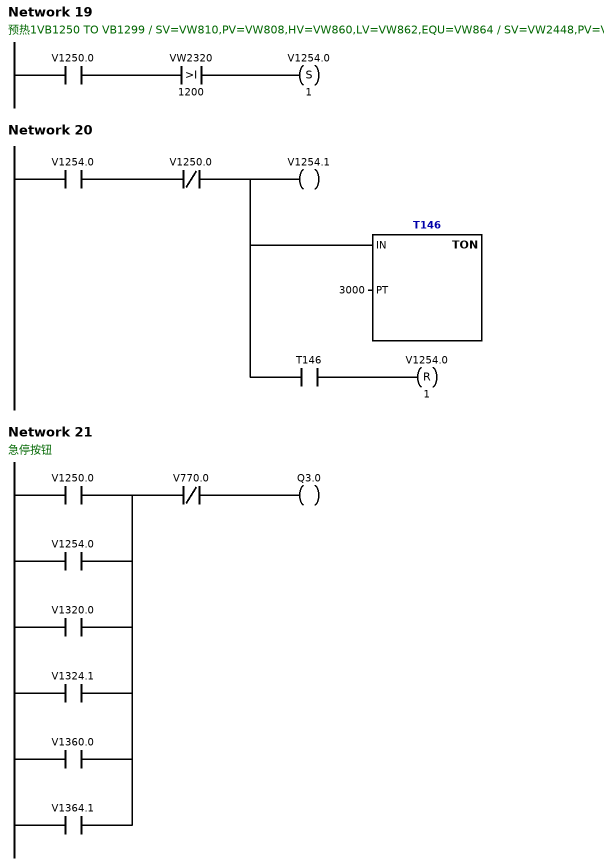
[picture p24: SBR4 networks 19-21]
Network 19
// 预热1VB1250 TO VB1299
// SV=VW810,PV=VW808,HV=VW860,LV=VW862,EQU=VW864
// SV=VW2448,PV=VW2320,HV=VW860,LV=VW862,EQU=VW864
// PV=VW2320 > 120 度就要冷却循环风关机
LD     V1250.0
AW>    VW2320, 1200
S      V1254.0, 1
Network 20
LD     V1254.0
AN     V1250.0
=      V1254.1
TON    T146, 3000
A      T146
R      V1254.0, 1
Network 21
// 急停按钮
LD     V1250.0
O      V1254.0
O      V1320.0
O      V1324.1
O      V1360.0
O      V1364.1
AN     V770.0
=      Q3.0
END_SUBROUTINE_BLOCK

SUBROUTINE_BLOCK WaveSpewWagVB1300_1319:SBR5
TITLE=WaveSpewWagVB1300_1319//T160_T164
BEGIN
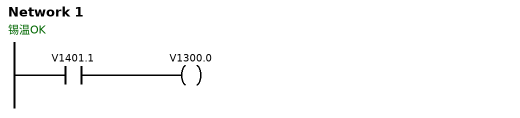
Network 1
// 锡温OK
LD     V1401.1
=      V1300.0
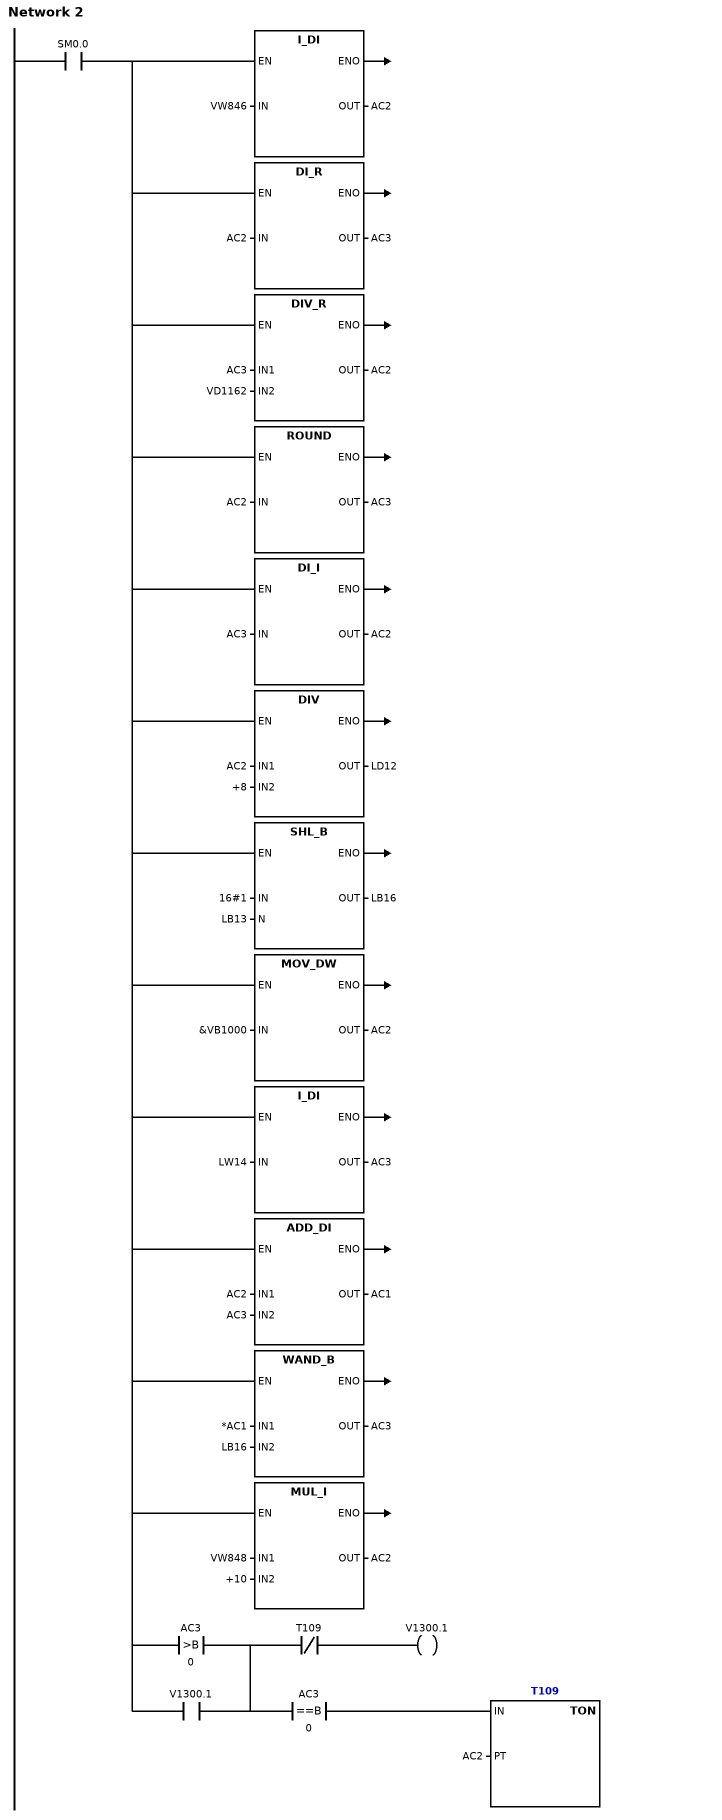
Network 2
LD     SM0.0
ITD    VW846, AC2
DTR    AC2, AC3
MOVR   AC3, AC2
/R     VD1162, AC2
ROUND  AC2, AC3
DTI    AC3, AC2
MOVW   AC2, LW14
DIV    +8, LD12
MOVB   16#1, LB16
SLB    LB16, LB13
MOVD   &VB1000, AC2
ITD    LW14, AC3
MOVD   AC2, AC1
+D     AC3, AC1
MOVB   *AC1, AC3
ANDB   LB16, AC3
MOVW   VW848, AC2
*I     +10, AC2
LDB>   AC3, 0
O      V1300.1
ALD
LPS
AN     T109
=      V1300.1
LPP
AB=    AC3, 0
TON    T109, AC2
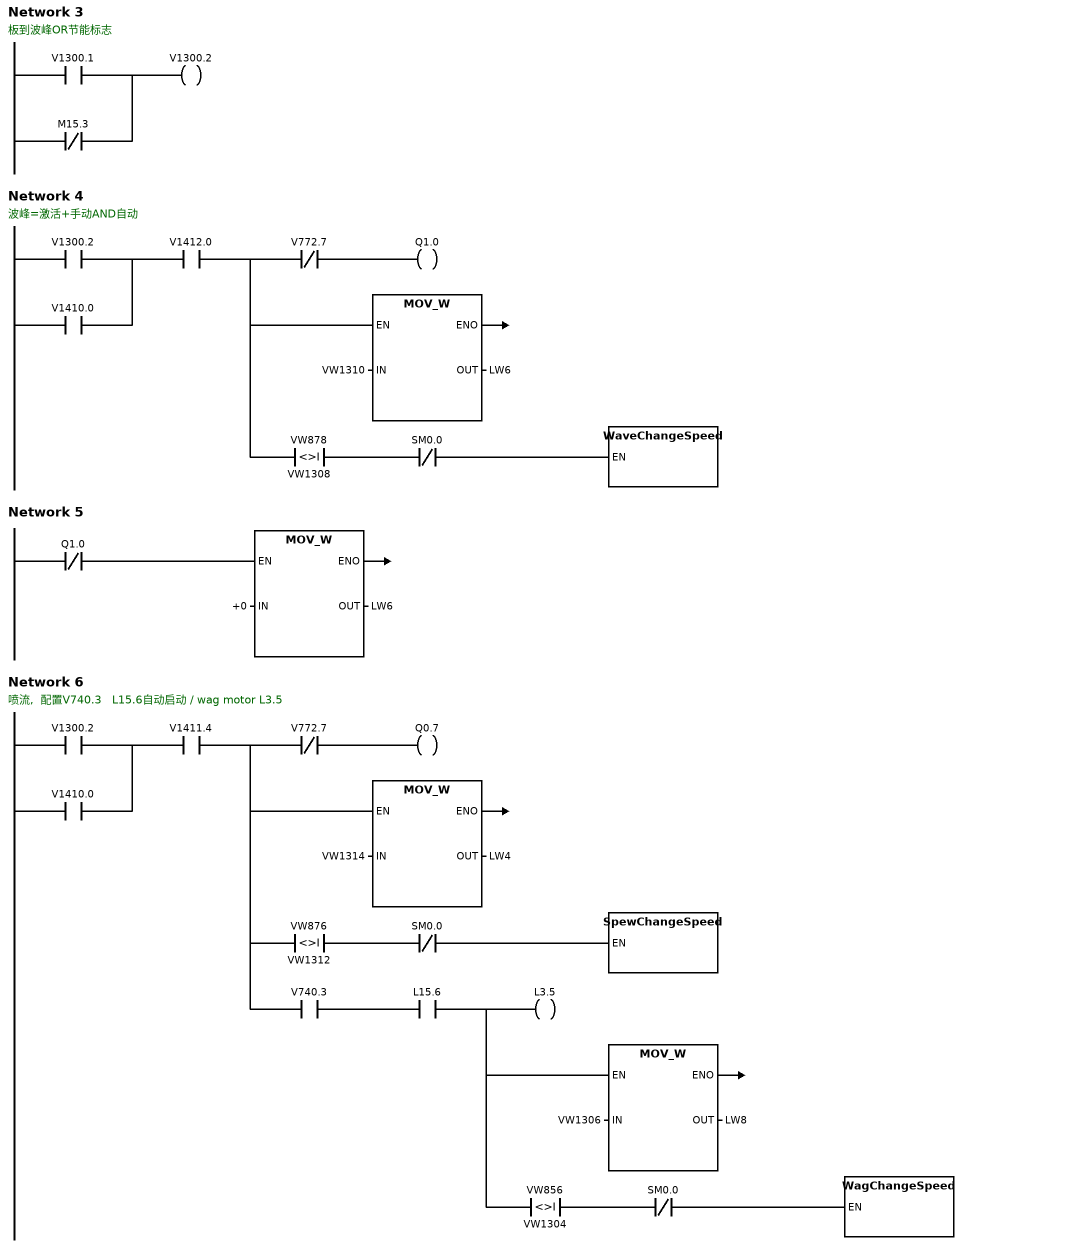
Network 3
// 板到波峰OR节能标志
LD     V1300.1
ON     M15.3
=      V1300.2
Network 4
// 波峰=激活+手动AND自动
LD     V1300.2
O      V1410.0
A      V1412.0
LPS
AN     V772.7
=      Q1.0
LRD
MOVW   VW1310, LW6
LPP
AW<>   VW878, VW1308
AN     SM0.0
CALL   WaveChangeSpeed:SBR23
Network 5
LDN    Q1.0
MOVW   +0, LW6
Network 6
// 喷流,  配置V740.3   L15.6自动启动
// wag motor L3.5
LD     V1300.2
O      V1410.0
A      V1411.4
LPS
AN     V772.7
=      Q0.7
LRD
MOVW   VW1314, LW4
LRD
AW<>   VW876, VW1312
AN     SM0.0
CALL   SpewChangeSpeed:SBR24
LPP
A      V740.3
A      L15.6
=      L3.5
MOVW   VW1306, LW8
AW<>   VW856, VW1304
AN     SM0.0
CALL   WagChangeSpeed:SBR22
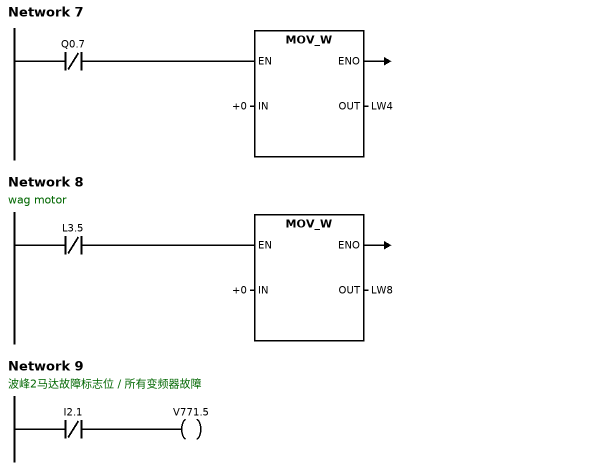
Network 7
LDN    Q0.7
MOVW   +0, LW4
Network 8
// wag motor 
LDN    L3.5
MOVW   +0, LW8
Network 9
// 波峰2马达故障标志位
// 所有变频器故障
LDN    I2.1
=      V771.5
Network 10
// 只要你配置了,喷流就可能产生故障标志位
Network 11
// 只要你配置了,摇动就可能产生故障标志位
END_SUBROUTINE_BLOCK

SUBROUTINE_BLOCK Preheat2VB1320_1359:SBR6
TITLE=
BEGIN
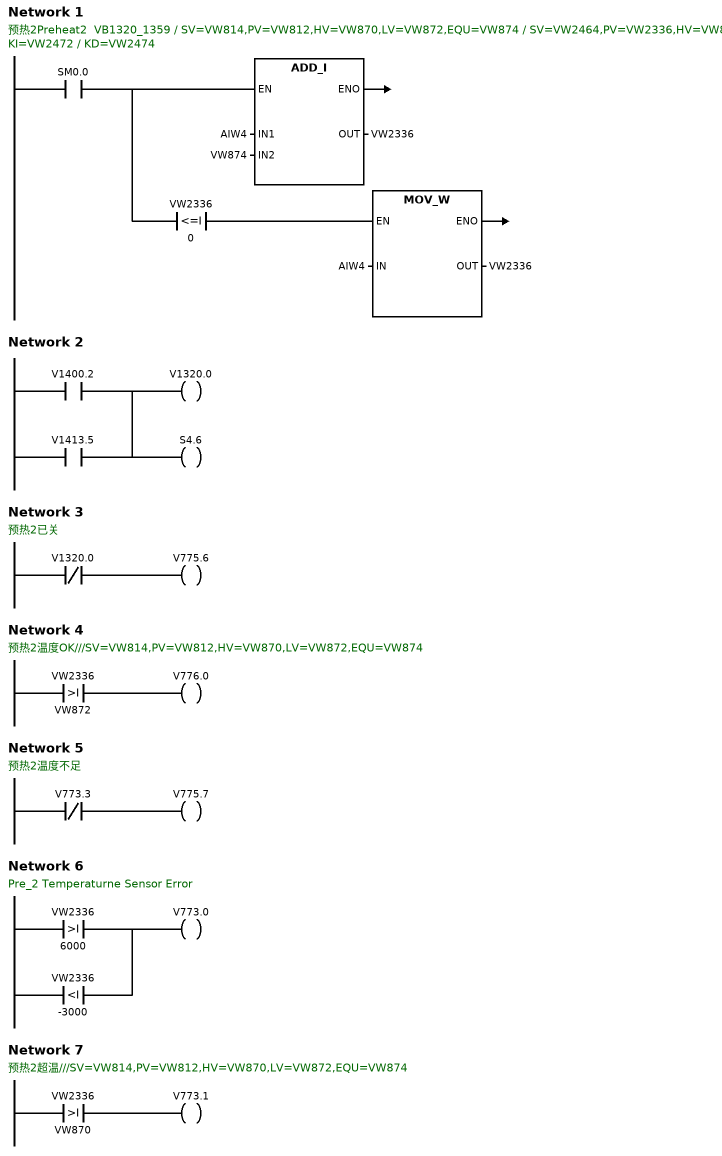
Network 1
// 预热2Preheat2  VB1320_1359
// SV=VW814,PV=VW812,HV=VW870,LV=VW872,EQU=VW874
// SV=VW2464,PV=VW2336,HV=VW870,LV=VW872,EQU=VW874
// 
// KT=VW2468
// KP=VW2470
// KI=VW2472
// KD=VW2474
LD     SM0.0
MOVW   AIW4, VW2336
+I     VW874, VW2336
AW<=   VW2336, 0
MOVW   AIW4, VW2336
Network 2
LD     V1400.2
O      V1413.5
=      V1320.0
=      S4.6
Network 3
// 预热2已关
LDN    V1320.0
=      V775.6
Network 4
// 预热2温度OK///SV=VW814,PV=VW812,HV=VW870,LV=VW872,EQU=VW874
LDW>   VW2336, VW872
=      V776.0
Network 5
// 预热2温度不足
LDN    V773.3
=      V775.7
Network 6
// Pre_2 Temperaturne Sensor Error
LDW>   VW2336, 6000
OW<    VW2336, -3000
=      V773.0
Network 7
// 预热2超温///SV=VW814,PV=VW812,HV=VW870,LV=VW872,EQU=VW874
LDW>   VW2336, VW870
=      V773.1
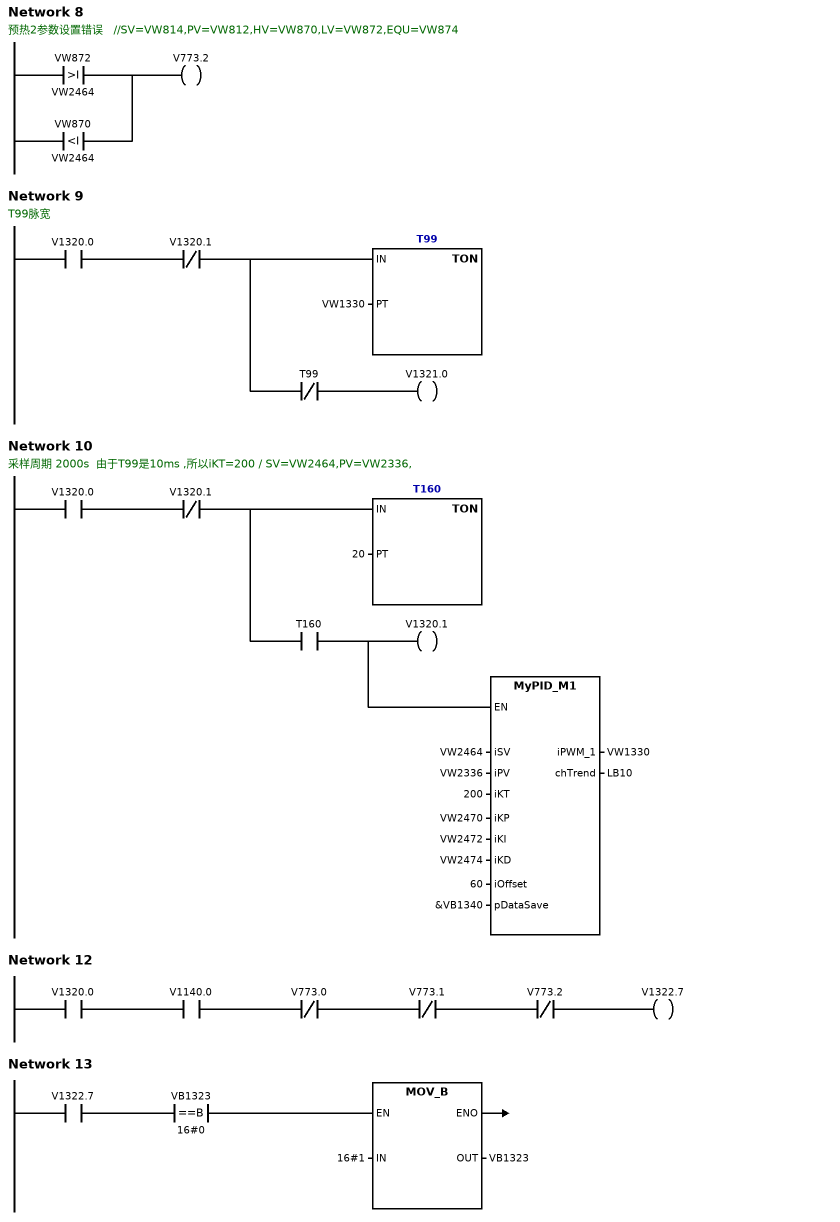
Network 8
// 预热2参数设置错误   //SV=VW814,PV=VW812,HV=VW870,LV=VW872,EQU=VW874
LDW>   VW872, VW2464
OW<    VW870, VW2464
=      V773.2
Network 9
// T99脉宽
LD     V1320.0
AN     V1320.1
TON    T99, VW1330
AN     T99
=      V1321.0
Network 10
// 采样周期 2000s  由于T99是10ms ,所以iKT=200
// SV=VW2464,PV=VW2336,
LD     V1320.0
AN     V1320.1
TON    T160, 20
A      T160
=      V1320.1
CALL   MyPID_M1:SBR30, VW2464, VW2336, 200, VW2470, VW2472, VW2474, 60, &VB1340, VW1330, LB10
Network 12
LD     V1320.0
A      V1140.0
AN     V773.0
AN     V773.1
AN     V773.2
=      V1322.7
Network 13
LD     V1322.7
AB=    VB1323, 16#0
MOVB   16#1, VB1323
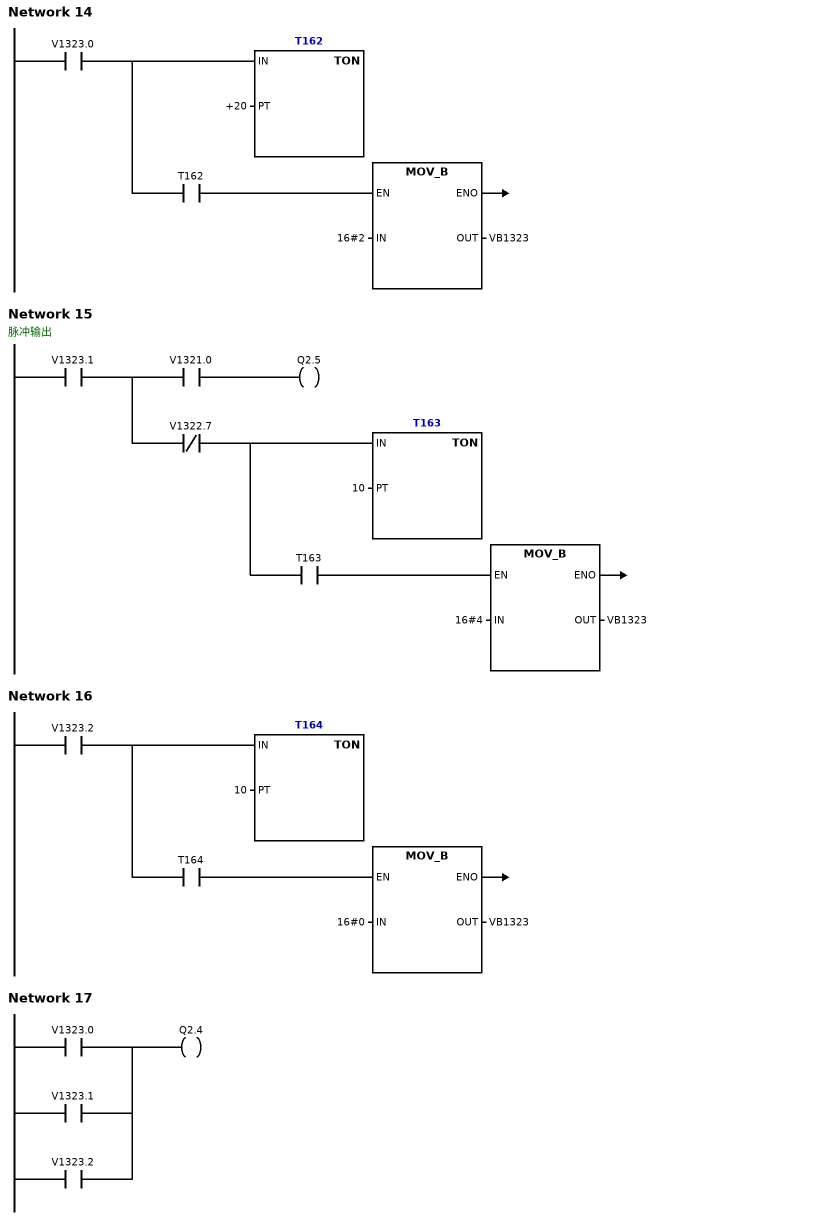
Network 14
LD     V1323.0
TON    T162, +20
A      T162
MOVB   16#2, VB1323
Network 15
// 脉冲输出
LD     V1323.1
LPS
A      V1321.0
=      Q2.5
LPP
AN     V1322.7
TON    T163, 10
A      T163
MOVB   16#4, VB1323
Network 16
LD     V1323.2
TON    T164, 10
A      T164
MOVB   16#0, VB1323
Network 17
LD     V1323.0
O      V1323.1
O      V1323.2
=      Q2.4
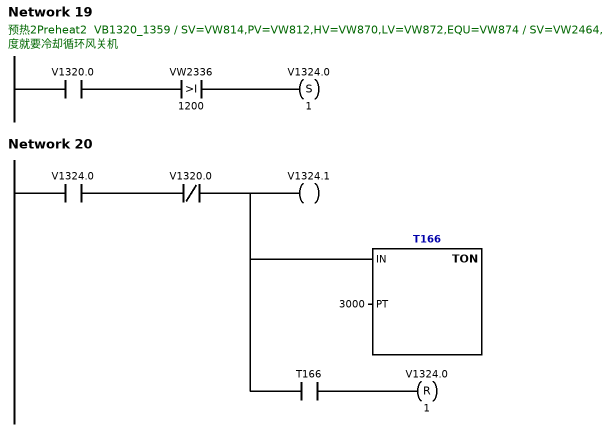
Network 19
// 预热2Preheat2  VB1320_1359
// SV=VW814,PV=VW812,HV=VW870,LV=VW872,EQU=VW874
// SV=VW2464,PV=VW2336,HV=VW870,LV=VW872,EQU=VW874
// PV=VW2336  >120 度就要冷却循环风关机
LD     V1320.0
AW>    VW2336, 1200
S      V1324.0, 1
Network 20
LD     V1324.0
AN     V1320.0
=      V1324.1
TON    T166, 3000
A      T166
R      V1324.0, 1
END_SUBROUTINE_BLOCK

SUBROUTINE_BLOCK Preheat3VB1360_1399:SBR7
TITLE=
BEGIN
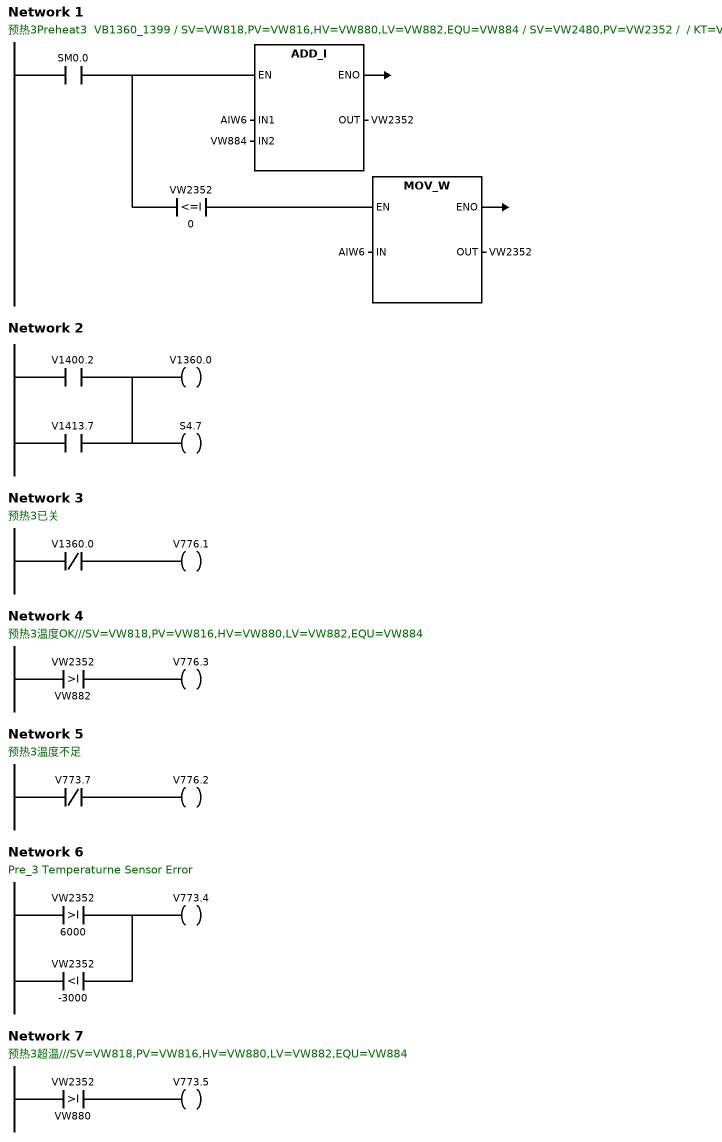
Network 1
// 预热3Preheat3  VB1360_1399
// SV=VW818,PV=VW816,HV=VW880,LV=VW882,EQU=VW884
// SV=VW2480,PV=VW2352
// 
// KT=VW2484=2s
// KP=VW2486
// KI=VW2488
// KD=VW2490
LD     SM0.0
MOVW   AIW6, VW2352
+I     VW884, VW2352
AW<=   VW2352, 0
MOVW   AIW6, VW2352
Network 2
LD     V1400.2
O      V1413.7
=      V1360.0
=      S4.7
Network 3
// 预热3已关
LDN    V1360.0
=      V776.1
Network 4
// 预热3温度OK///SV=VW818,PV=VW816,HV=VW880,LV=VW882,EQU=VW884
LDW>   VW2352, VW882
=      V776.3
Network 5
// 预热3温度不足
LDN    V773.7
=      V776.2
Network 6
// Pre_3 Temperaturne Sensor Error
LDW>   VW2352, 6000
OW<    VW2352, -3000
=      V773.4
Network 7
// 预热3超温///SV=VW818,PV=VW816,HV=VW880,LV=VW882,EQU=VW884
LDW>   VW2352, VW880
=      V773.5
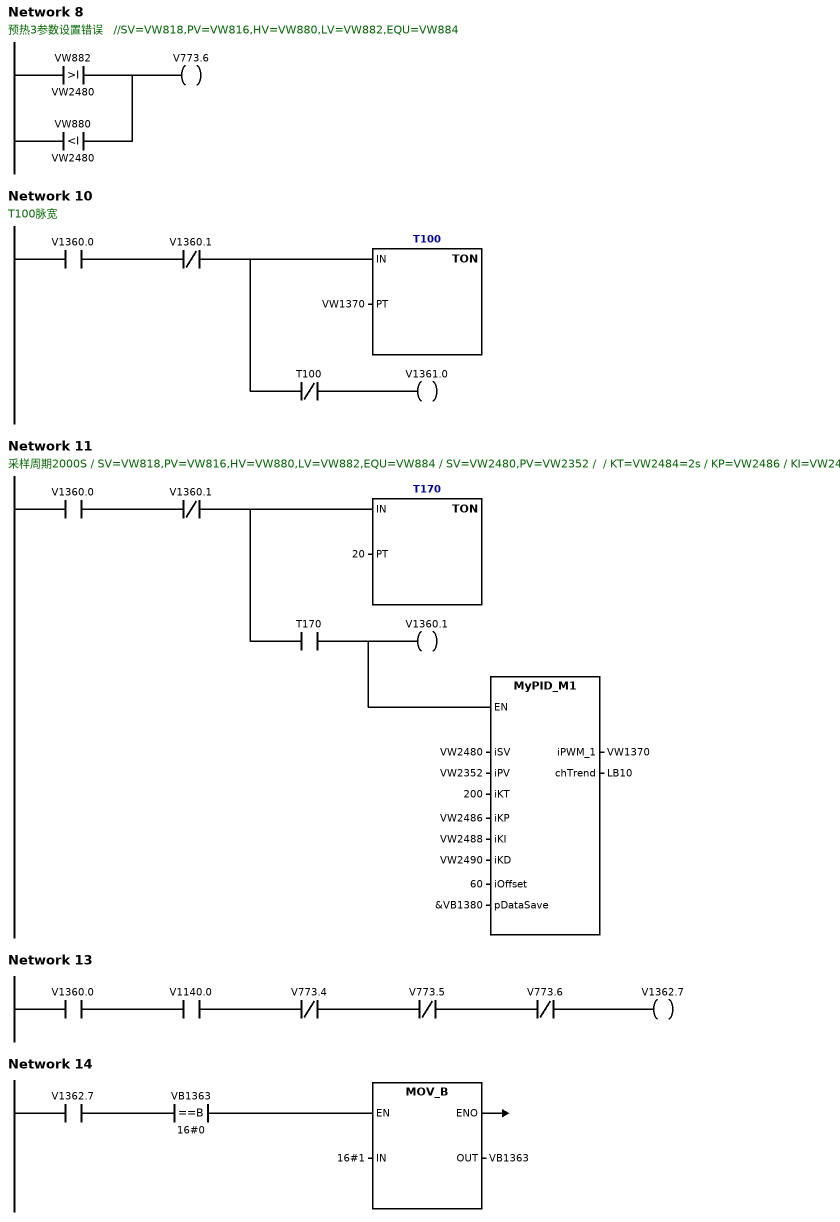
Network 8
// 预热3参数设置错误   //SV=VW818,PV=VW816,HV=VW880,LV=VW882,EQU=VW884
LDW>   VW882, VW2480
OW<    VW880, VW2480
=      V773.6
Network 10
// T100脉宽
LD     V1360.0
AN     V1360.1
TON    T100, VW1370
AN     T100
=      V1361.0
Network 11
// 采样周期2000S
// SV=VW818,PV=VW816,HV=VW880,LV=VW882,EQU=VW884
// SV=VW2480,PV=VW2352
// 
// KT=VW2484=2s
// KP=VW2486
// KI=VW2488
// KD=VW2490
LD     V1360.0
AN     V1360.1
TON    T170, 20
A      T170
=      V1360.1
CALL   MyPID_M1:SBR30, VW2480, VW2352, 200, VW2486, VW2488, VW2490, 60, &VB1380, VW1370, LB10
Network 13
LD     V1360.0
A      V1140.0
AN     V773.4
AN     V773.5
AN     V773.6
=      V1362.7
Network 14
LD     V1362.7
AB=    VB1363, 16#0
MOVB   16#1, VB1363
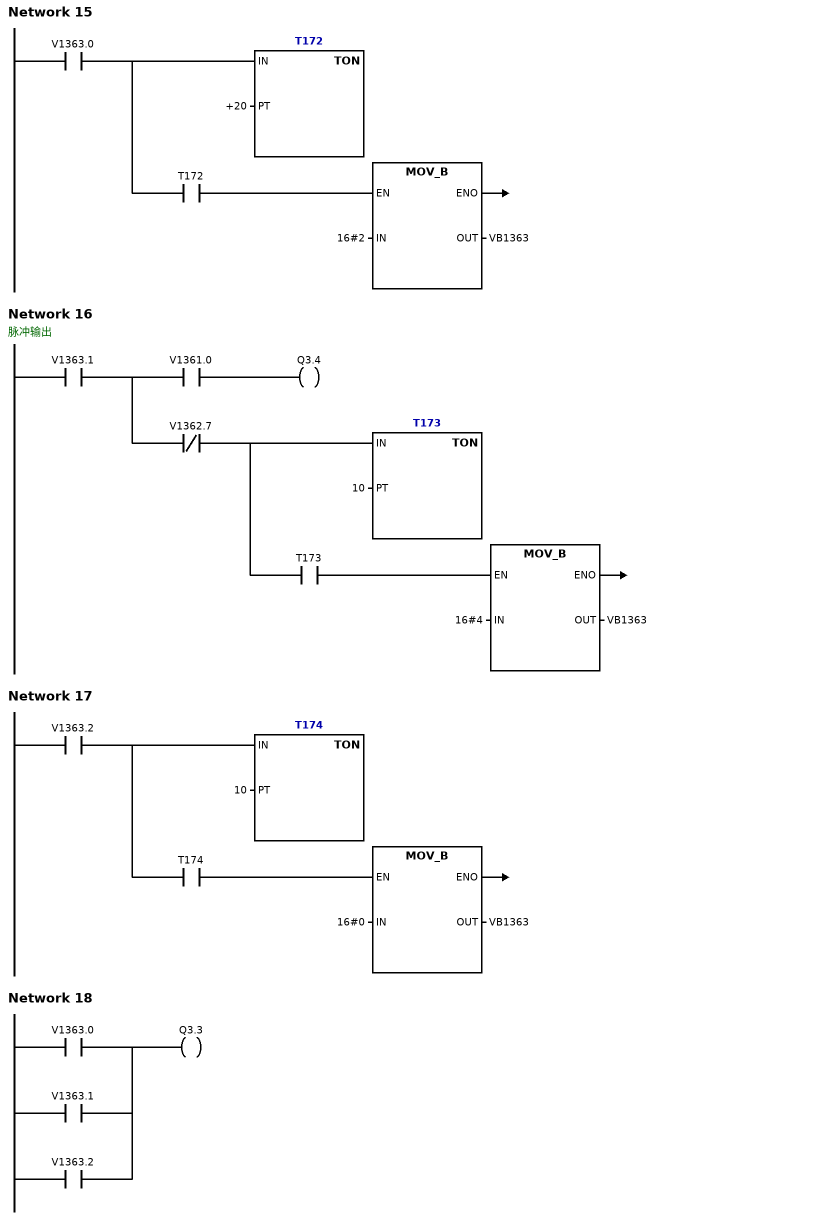
Network 15
LD     V1363.0
TON    T172, +20
A      T172
MOVB   16#2, VB1363
Network 16
// 脉冲输出
LD     V1363.1
LPS
A      V1361.0
=      Q3.4
LPP
AN     V1362.7
TON    T173, 10
A      T173
MOVB   16#4, VB1363
Network 17
LD     V1363.2
TON    T174, 10
A      T174
MOVB   16#0, VB1363
Network 18
LD     V1363.0
O      V1363.1
O      V1363.2
=      Q3.3
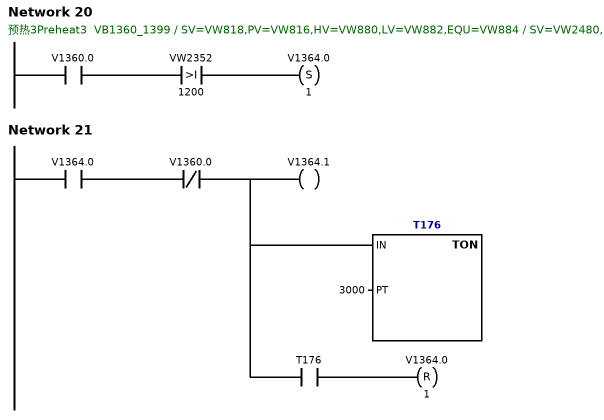
Network 20
// 预热3Preheat3  VB1360_1399
// SV=VW818,PV=VW816,HV=VW880,LV=VW882,EQU=VW884
// SV=VW2480,PV=VW2352
// PV=VW2352  >120 度就要冷却循环风关机
LD     V1360.0
AW>    VW2352, 1200
S      V1364.0, 1
Network 21
LD     V1364.0
AN     V1360.0
=      V1364.1
TON    T176, 3000
A      T176
R      V1364.0, 1
END_SUBROUTINE_BLOCK

SUBROUTINE_BLOCK AutoVB1400_1409:SBR8
TITLE=AutoVB1400_1409
BEGIN
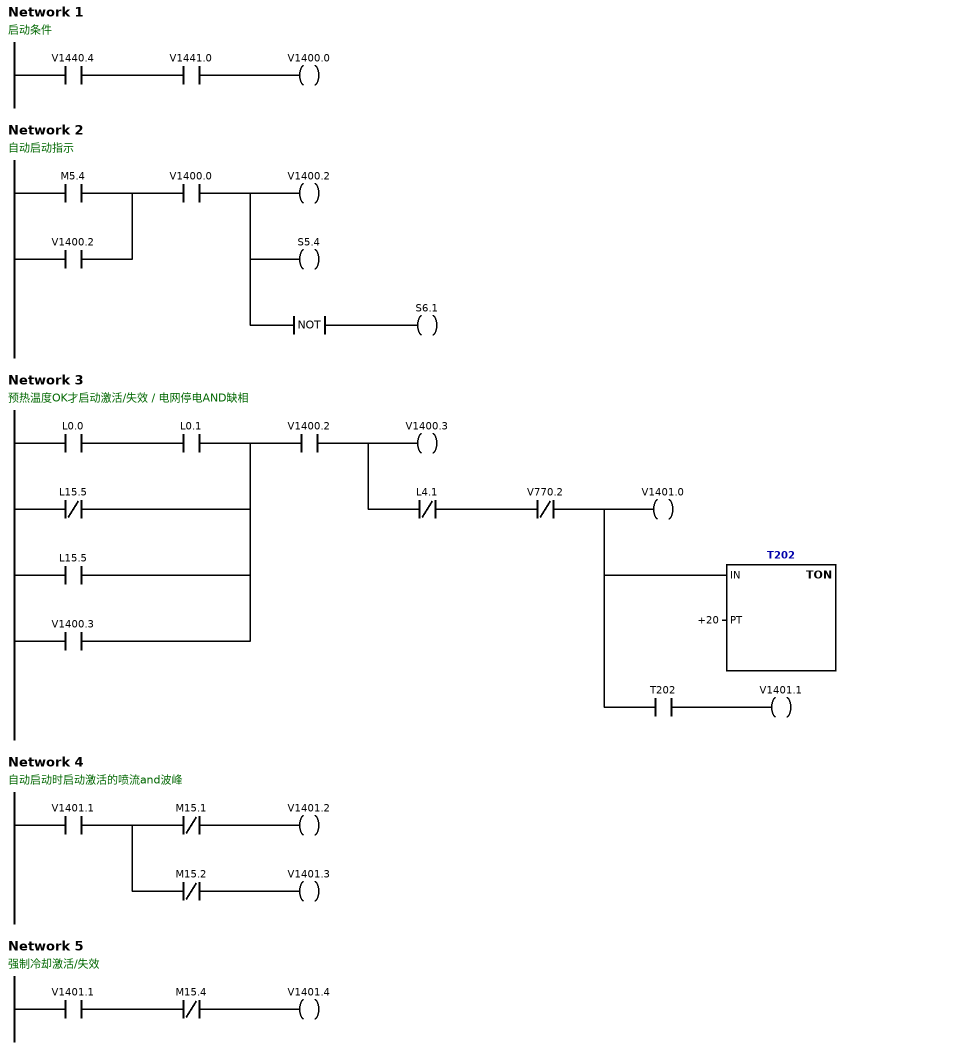
Network 1
// 启动条件
LD     V1440.4
A      V1441.0
=      V1400.0
Network 2
// 自动启动指示
LD     M5.4
O      V1400.2
A      V1400.0
=      V1400.2
=      S5.4
NOT
=      S6.1
Network 3
// 预热温度OK才启动激活/失效
// 电网停电AND缺相
LD     L0.0
A      L0.1
ON     L15.5
O      L15.5
O      V1400.3
A      V1400.2
=      V1400.3
AN     L4.1
AN     V770.2
=      V1401.0
TON    T202, +20
A      T202
=      V1401.1
Network 4
// 自动启动时启动激活的喷流and波峰
LD     V1401.1
LPS
AN     M15.1
=      V1401.2
LPP
AN     M15.2
=      V1401.3
Network 5
// 强制冷却激活/失效
LD     V1401.1
AN     M15.4
=      V1401.4
END_SUBROUTINE_BLOCK

SUBROUTINE_BLOCK ManualVB1410_VB1439:SBR9
TITLE=ManualVB1410_VB1439lhy69698
BEGIN
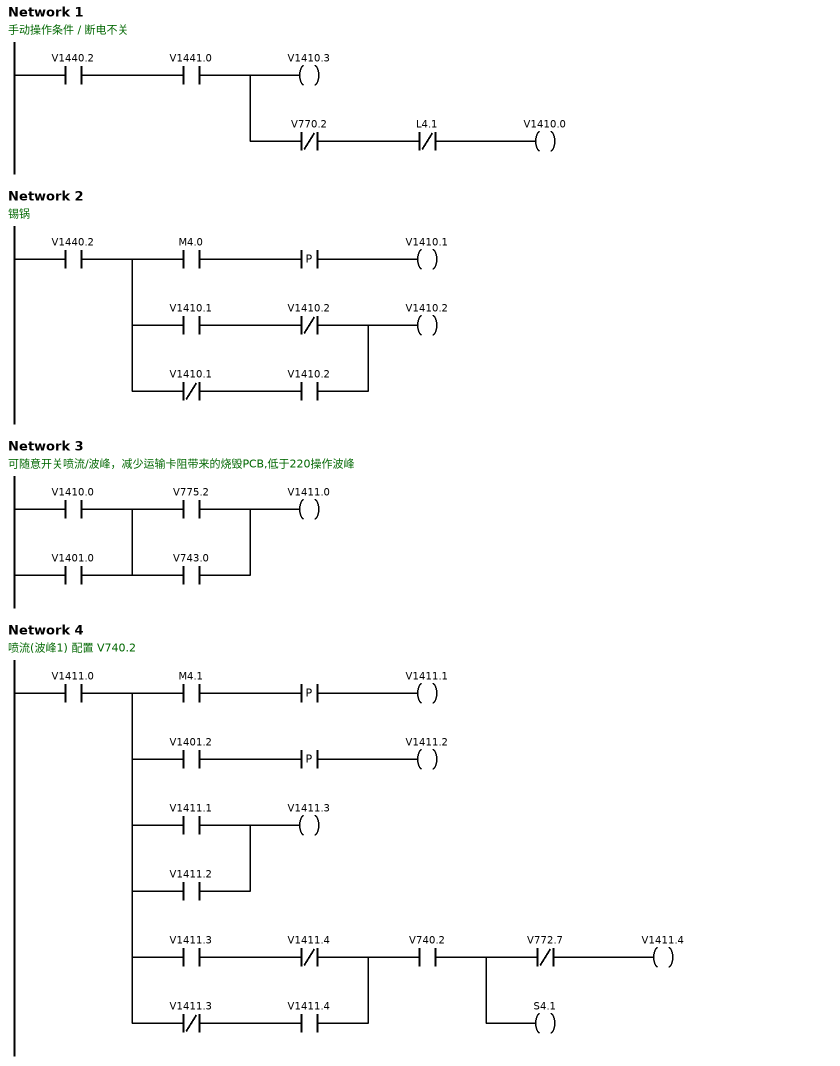
Network 1
// 手动操作条件
// 断电不关
LD     V1440.2
A      V1441.0
=      V1410.3
AN     V770.2
AN     L4.1
=      V1410.0
Network 2
// 锡锅
LD     V1440.2
LPS
A      M4.0
EU
=      V1410.1
LPP
LD     V1410.1
AN     V1410.2
LDN    V1410.1
A      V1410.2
OLD
ALD
=      V1410.2
Network 3
// 可随意开关喷流/波峰，减少运输卡阻带来的烧毁PCB,低于220操作波峰
LD     V1410.0
O      V1401.0
LD     V775.2
O      V743.0
ALD
=      V1411.0
Network 4
// 喷流(波峰1) 配置 V740.2 
LD     V1411.0
LPS
A      M4.1
EU
=      V1411.1
LRD
A      V1401.2
EU
=      V1411.2
LRD
LD     V1411.1
O      V1411.2
ALD
=      V1411.3
LPP
LD     V1411.3
AN     V1411.4
LDN    V1411.3
A      V1411.4
OLD
A      V740.2
ALD
LPS
AN     V772.7
=      V1411.4
LPP
=      S4.1
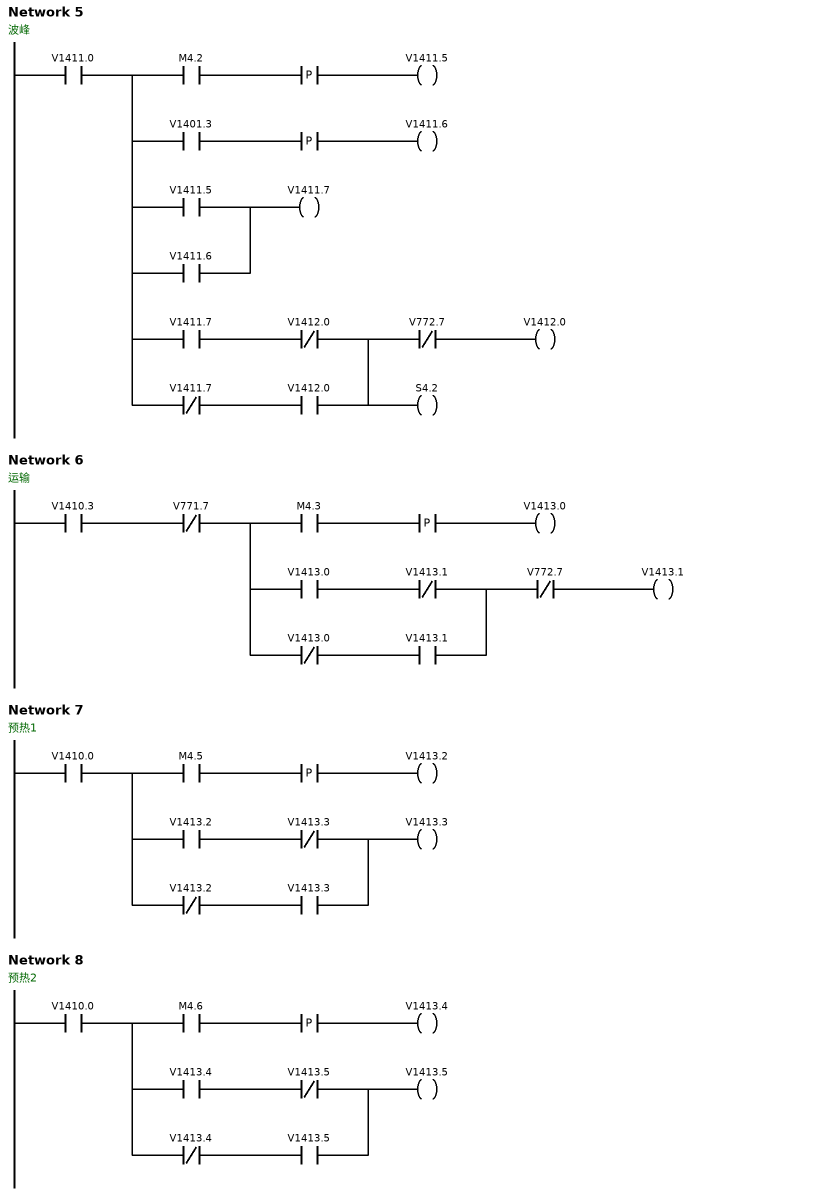
Network 5
// 波峰
LD     V1411.0
LPS
A      M4.2
EU
=      V1411.5
LRD
A      V1401.3
EU
=      V1411.6
LRD
LD     V1411.5
O      V1411.6
ALD
=      V1411.7
LPP
LD     V1411.7
AN     V1412.0
LDN    V1411.7
A      V1412.0
OLD
ALD
LPS
AN     V772.7
=      V1412.0
LPP
=      S4.2
Network 6
// 运输
LD     V1410.3
AN     V771.7
LPS
A      M4.3
EU
=      V1413.0
LPP
LD     V1413.0
AN     V1413.1
LDN    V1413.0
A      V1413.1
OLD
ALD
AN     V772.7
=      V1413.1
Network 7
// 预热1
LD     V1410.0
LPS
A      M4.5
EU
=      V1413.2
LPP
LD     V1413.2
AN     V1413.3
LDN    V1413.2
A      V1413.3
OLD
ALD
=      V1413.3
Network 8
// 预热2
LD     V1410.0
LPS
A      M4.6
EU
=      V1413.4
LPP
LD     V1413.4
AN     V1413.5
LDN    V1413.4
A      V1413.5
OLD
ALD
=      V1413.5
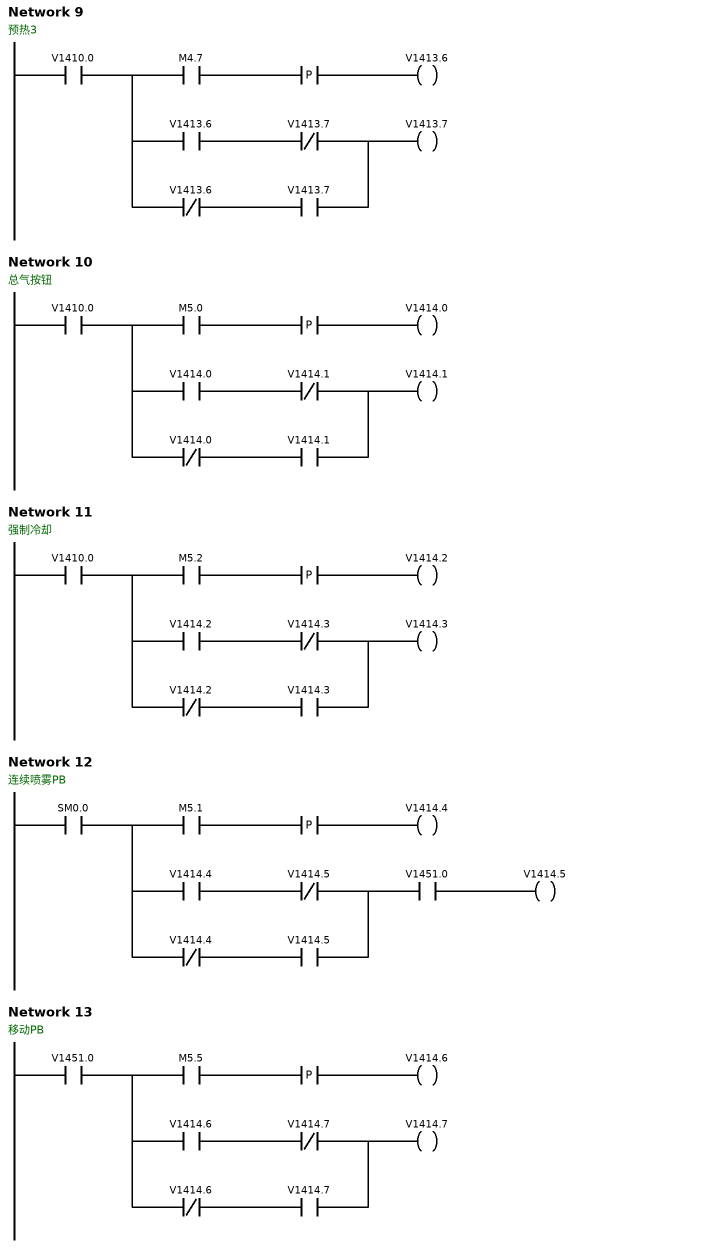
Network 9
// 预热3
LD     V1410.0
LPS
A      M4.7
EU
=      V1413.6
LPP
LD     V1413.6
AN     V1413.7
LDN    V1413.6
A      V1413.7
OLD
ALD
=      V1413.7
Network 10
// 总气按钮
LD     V1410.0
LPS
A      M5.0
EU
=      V1414.0
LPP
LD     V1414.0
AN     V1414.1
LDN    V1414.0
A      V1414.1
OLD
ALD
=      V1414.1
Network 11
// 强制冷却
LD     V1410.0
LPS
A      M5.2
EU
=      V1414.2
LPP
LD     V1414.2
AN     V1414.3
LDN    V1414.2
A      V1414.3
OLD
ALD
=      V1414.3
Network 12
// 连续喷雾PB
LD     SM0.0
LPS
A      M5.1
EU
=      V1414.4
LPP
LD     V1414.4
AN     V1414.5
LDN    V1414.4
A      V1414.5
OLD
ALD
A      V1451.0
=      V1414.5
Network 13
// 移动PB
LD     V1451.0
LPS
A      M5.5
EU
=      V1414.6
LPP
LD     V1414.6
AN     V1414.7
LDN    V1414.6
A      V1414.7
OLD
ALD
=      V1414.7
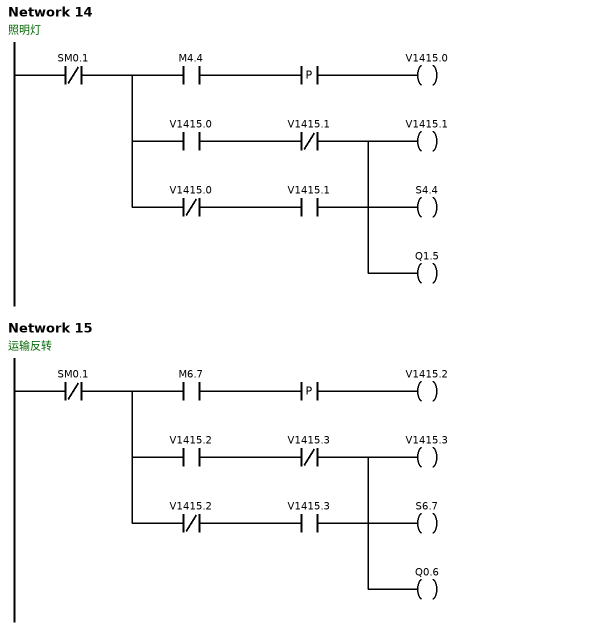
Network 14
// 照明灯
LDN    SM0.1
LPS
A      M4.4
EU
=      V1415.0
LPP
LD     V1415.0
AN     V1415.1
LDN    V1415.0
A      V1415.1
OLD
ALD
=      V1415.1
=      S4.4
=      Q1.5
Network 15
// 运输反转
LDN    SM0.1
LPS
A      M6.7
EU
=      V1415.2
LPP
LD     V1415.2
AN     V1415.3
LDN    V1415.2
A      V1415.3
OLD
ALD
=      V1415.3
=      S6.7
=      Q0.6
END_SUBROUTINE_BLOCK

SUBROUTINE_BLOCK SprayMoveVB1500_VB1649:SBR10
TITLE=SprayMoveVB1500_1649
BEGIN
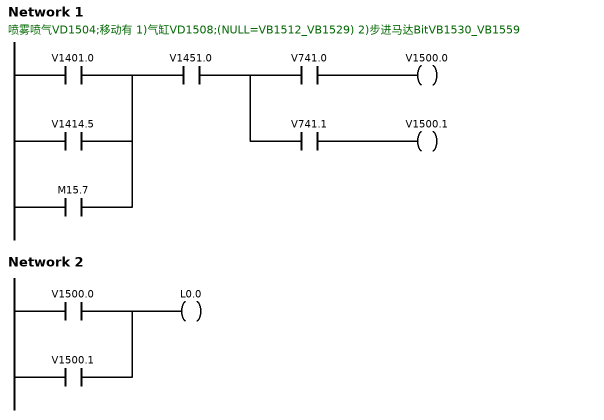
Network 1
// 喷雾喷气VD1504;移动有 1)气缸VD1508;(NULL=VB1512_VB1529) 2)步进马达BitVB1530_VB1559
LD     V1401.0
O      V1414.5
O      M15.7
A      V1451.0
LPS
A      V741.0
=      V1500.0
LPP
A      V741.1
=      V1500.1
Network 2
LD     V1500.0
O      V1500.1
=      L0.0
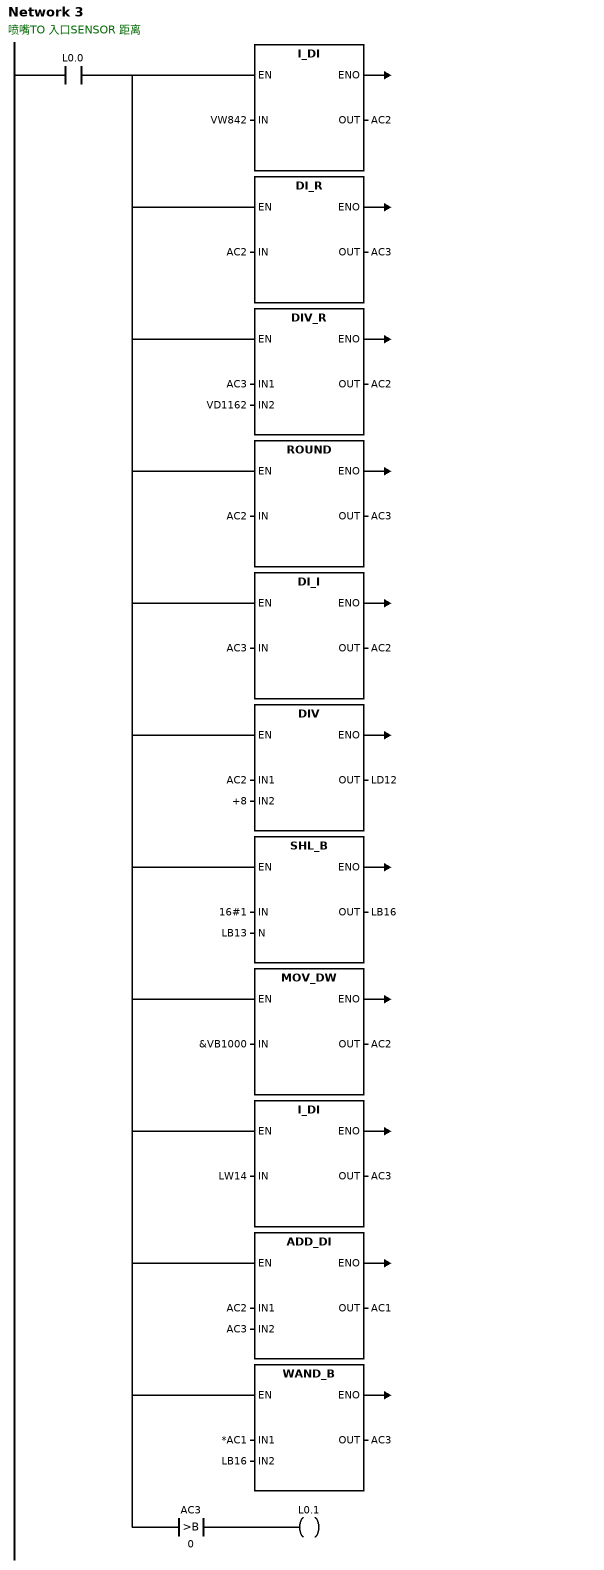
Network 3
// 喷嘴TO 入口SENSOR 距离
LD     L0.0
ITD    VW842, AC2
DTR    AC2, AC3
MOVR   AC3, AC2
/R     VD1162, AC2
ROUND  AC2, AC3
DTI    AC3, AC2
MOVW   AC2, LW14
DIV    +8, LD12
MOVB   16#1, LB16
SLB    LB16, LB13
MOVD   &VB1000, AC2
ITD    LW14, AC3
MOVD   AC2, AC1
+D     AC3, AC1
MOVB   *AC1, AC3
ANDB   LB16, AC3
AB>    AC3, 0
=      L0.1
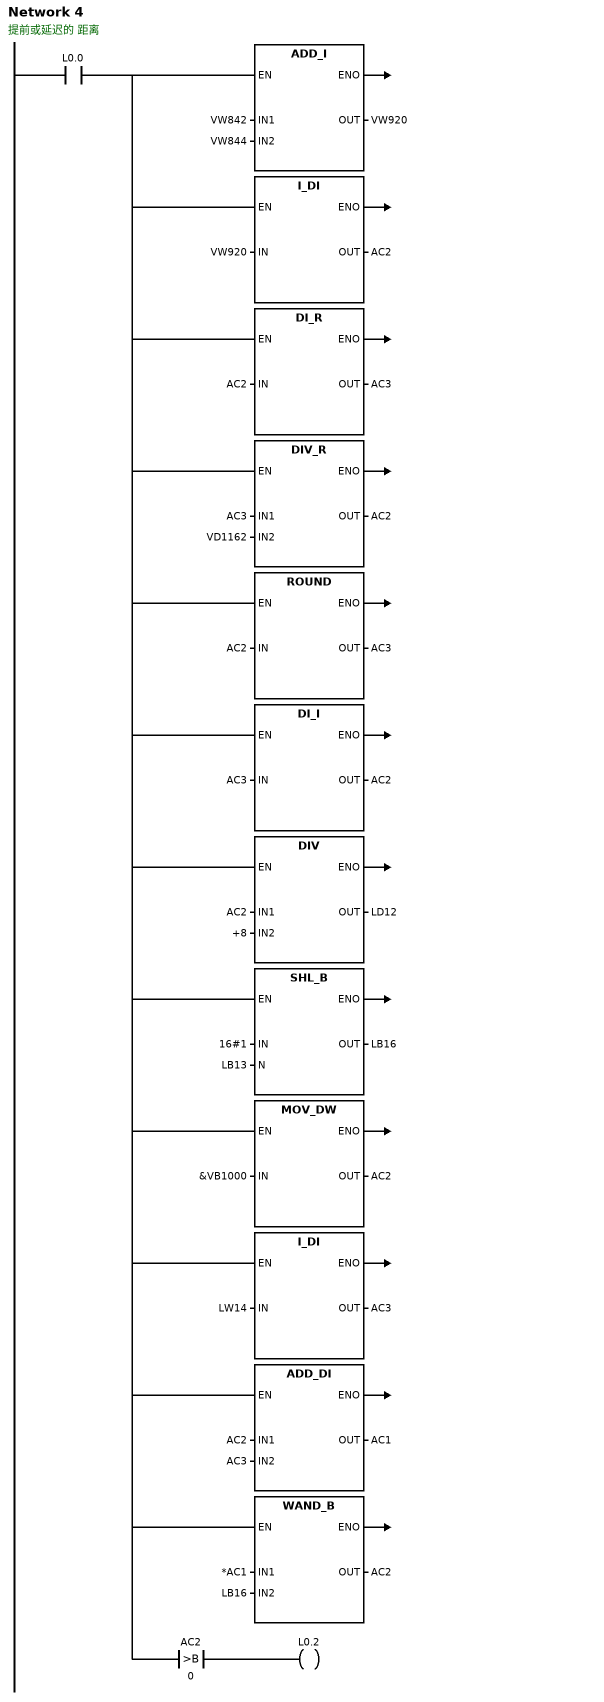
Network 4
// 提前或延迟的 距离
LD     L0.0
MOVW   VW842, VW920
+I     VW844, VW920
ITD    VW920, AC2
DTR    AC2, AC3
MOVR   AC3, AC2
/R     VD1162, AC2
ROUND  AC2, AC3
DTI    AC3, AC2
MOVW   AC2, LW14
DIV    +8, LD12
MOVB   16#1, LB16
SLB    LB16, LB13
MOVD   &VB1000, AC2
ITD    LW14, AC3
MOVD   AC2, AC1
+D     AC3, AC1
MOVB   *AC1, AC2
ANDB   LB16, AC2
AB>    AC2, 0
=      L0.2
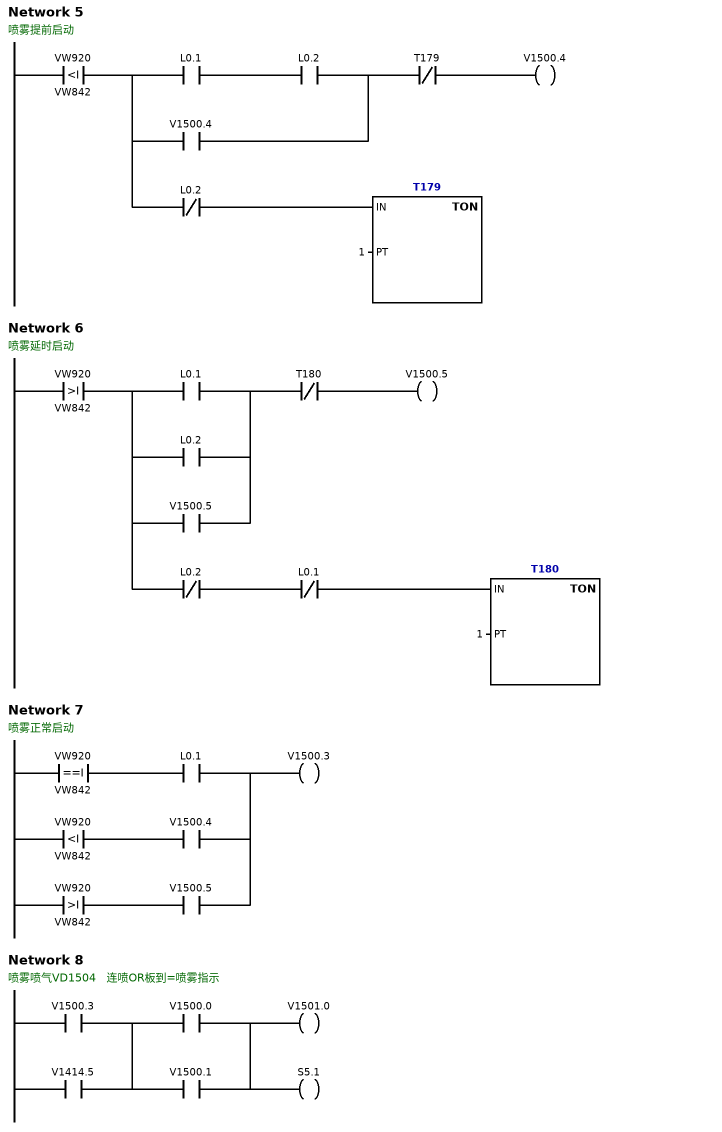
Network 5
// 喷雾提前启动
LDW<   VW920, VW842
LPS
LD     L0.1
A      L0.2
O      V1500.4
ALD
AN     T179
=      V1500.4
LPP
AN     L0.2
TON    T179, 1
Network 6
// 喷雾延时启动
LDW>   VW920, VW842
LPS
LD     L0.1
O      L0.2
O      V1500.5
ALD
AN     T180
=      V1500.5
LPP
AN     L0.2
AN     L0.1
TON    T180, 1
Network 7
// 喷雾正常启动
LDW=   VW920, VW842
A      L0.1
LDW<   VW920, VW842
A      V1500.4
OLD
LDW>   VW920, VW842
A      V1500.5
OLD
=      V1500.3
Network 8
// 喷雾喷气VD1504   连喷OR板到=喷雾指示
LD     V1500.3
O      V1414.5
LD     V1500.0
O      V1500.1
ALD
=      V1501.0
=      S5.1
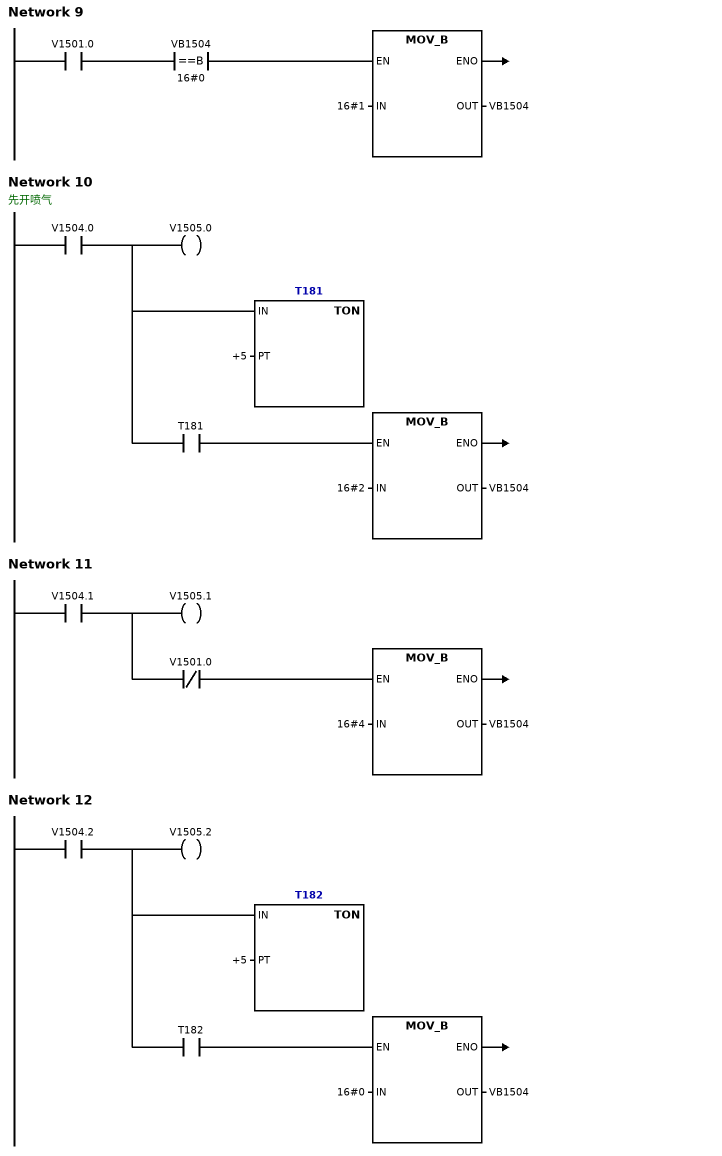
Network 9
LD     V1501.0
AB=    VB1504, 16#0
MOVB   16#1, VB1504
Network 10
// 先开喷气
LD     V1504.0
=      V1505.0
TON    T181, +5
A      T181
MOVB   16#2, VB1504
Network 11
LD     V1504.1
=      V1505.1
AN     V1501.0
MOVB   16#4, VB1504
Network 12
LD     V1504.2
=      V1505.2
TON    T182, +5
A      T182
MOVB   16#0, VB1504
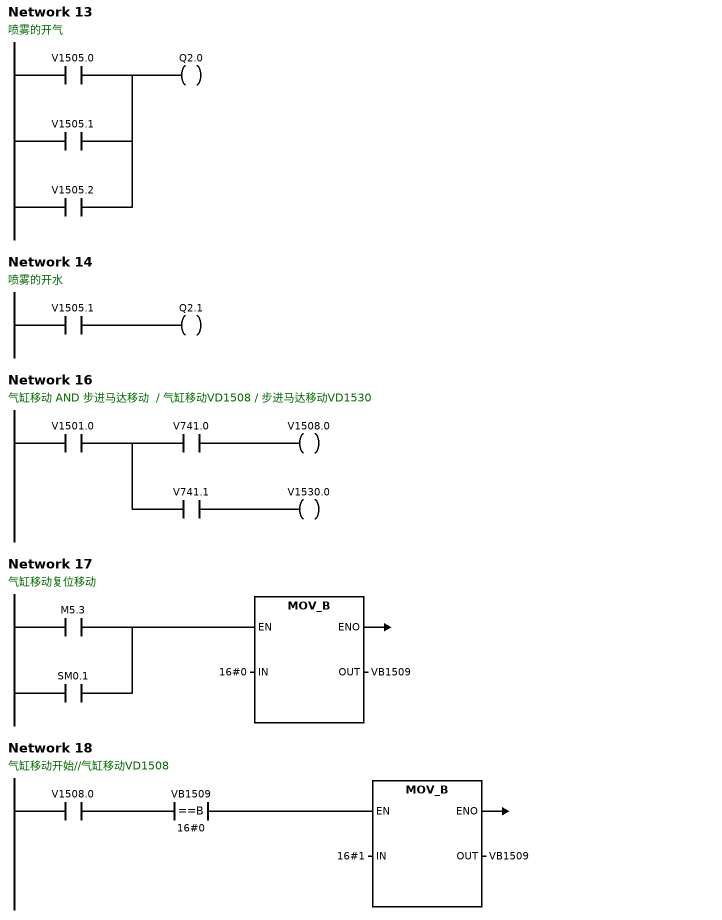
Network 13
// 喷雾的开气
LD     V1505.0
O      V1505.1
O      V1505.2
=      Q2.0
Network 14
// 喷雾的开水
LD     V1505.1
=      Q2.1
Network 16
// 气缸移动 AND 步进马达移动 
// 气缸移动VD1508
// 步进马达移动VD1530
LD     V1501.0
LPS
A      V741.0
=      V1508.0
LPP
A      V741.1
=      V1530.0
Network 17
// 气缸移动复位移动
LD     M5.3
O      SM0.1
MOVB   16#0, VB1509
Network 18
// 气缸移动开始//气缸移动VD1508
LD     V1508.0
AB=    VB1509, 16#0
MOVB   16#1, VB1509
